Staubli VAL3: ex12.pjx

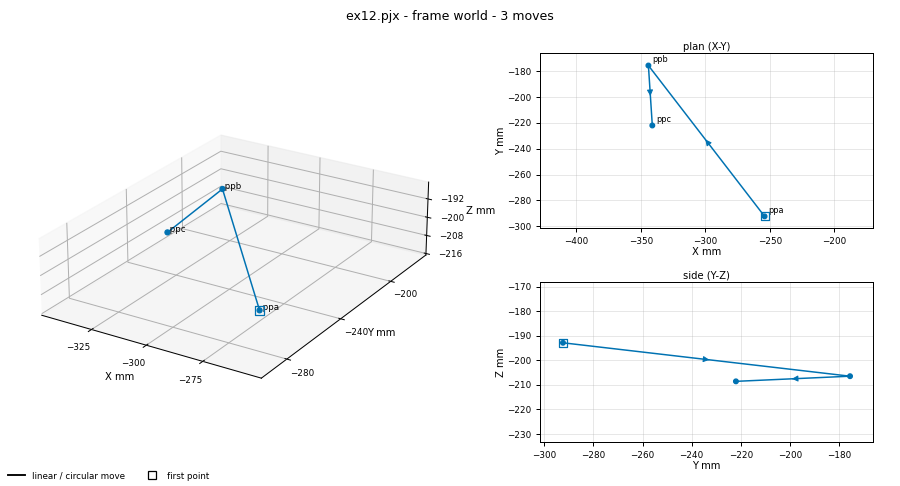
[picture p0: tool path of ex12.pjx in frame world, 3 of 5 moves have a stored position in this frame; points joined in program order, loops and branches not executed]
--- ex12.pjx ---
Parameters version=s7.4 stackSize=5000 millimeterUnit=true
Program file=ex12.pgx
Program file=start.pgx
Program file=stop.pgx
Data file=ex12.dtx

--- ex12.dtx ---
jointRx jdepart = {j1=-36.272631, j2=39.481199, j3=20.55017, j4=0.162735, j5=51.300785, j6=211.211358}
jointRx ppd = {j1=-87.396973, j2=33.472284, j3=31.213379, j4=-2.062683, j5=74.065576, j6=181.630117}
mdesc mNomSpeed
mdesc mlent = {accel=9, vel=30, decel=9, blend=off}
pointRx ppa = {x=-254.02593, y=-292.437944, z=-192.828909, rx=1.85447, ry=-179.679472, rz=-46.301311, fatherId=world[0]}
pointRx ppb = {x=-344.105703, y=-175.494959, z=-206.436129, rx=2.054021, ry=179.074214, rz=-24.317832, fatherId=world[0]}
pointRx ppc = {x=-341.079018, y=-221.979028, z=-208.532198, rx=2.924873, ry=178.271133, rz=-27.955909, fatherId=world[0]}
tool tstylo = {z=100, fatherId=flange[0], ioLink=valve1}

--- start.pgx ---
program start()
begin
  call ex12()
end

--- ex12.pgx ---
program ex12()
begin
  movej(jdepart,tstylo,mlent)
  movej(ppa,tstylo,mlent)
  movel(ppb,tstylo,mlent)
  movel(ppc,tstylo,mlent)
  movej(jdepart,tstylo,mlent)
  waitEndMove()
end
